// TwinCAT 3 PLC project PLC_Server_02
// ProgramVersion: 3.1.4023.0
// libraries:
//   Tc2_MC2, * (Beckhoff Automation GmbH)
//   Tc2_Standard, * (Beckhoff Automation GmbH)
//   Tc2_System, * (Beckhoff Automation GmbH)
//   Tc3_Module, * (Beckhoff Automation GmbH)
// project tree:
//   DUTs/ ST_Motor.TcDUT, ST_MotorCtrl.TcDUT
//   / GlobalTextList.TcGTLO, PlcTask.TcTTO, VISU_TASK.TcTTO
//   POUs/ FB_Math.TcPOU, MAIN.TcPOU
//   VISUs/ motor_status.TcVIS, VisualizationManager.TcVMO (not stored)
// real-time tasks:
//   TASK PlcTask: cycle T#10ms, priority 20, ADS port 350
//   TASK VISU_TASK: cycle T#200000us, priority 30, ADS port 351
// motion (NC):
//   TASK NC-Task 1 SAF: cycle T#2ms, priority 4, ADS port 501
//   TASK NC-Task 1 SVB: cycle T#10ms, priority 8, ADS port 511
//   AXIS Motor-0 (id 1)
//     OtherSettings: AllowMotionCmdToSlave=true
//     encoder EncType=1
//     drive DrvType=5
//       Analog: TorqueSetpointScale=10, ScaleFactorActTorque=0.1
//       TimeComp: TaskDelayCycles=1
//     controller CtrType=1
//       CtrPara: PriorControlFactor=1
//         Observer: BandWidth=20
//   AXIS Motor-1 (id 2)
//     OtherSettings: AllowMotionCmdToSlave=true
//     encoder EncType=1
//     drive DrvType=5
//       Analog: TorqueSetpointScale=10, ScaleFactorActTorque=0.1
//       TimeComp: TaskDelayCycles=1
//     controller CtrType=1
//       CtrPara: PriorControlFactor=1
//         Observer: BandWidth=20
//   AXIS Motor-2 (id 3)
//     OtherSettings: AllowMotionCmdToSlave=true
//     encoder EncType=1
//     drive DrvType=5
//       Analog: TorqueSetpointScale=10, ScaleFactorActTorque=0.1
//       TimeComp: TaskDelayCycles=1
//     controller CtrType=1
//       CtrPara: PriorControlFactor=1
//         Observer: BandWidth=20
//   AXIS Motor-3 (id 4)
//     OtherSettings: AllowMotionCmdToSlave=true
//     encoder EncType=1
//     drive DrvType=5
//       Analog: TorqueSetpointScale=10, ScaleFactorActTorque=0.1
//       TimeComp: TaskDelayCycles=1
//     controller CtrType=1
//       CtrPara: PriorControlFactor=1
//         Observer: BandWidth=20
//   AXIS Motor-4 (id 5)
//     OtherSettings: AllowMotionCmdToSlave=true
//     encoder EncType=1
//     drive DrvType=5
//       Analog: TorqueSetpointScale=10, ScaleFactorActTorque=0.1
//       TimeComp: TaskDelayCycles=1
//     controller CtrType=1
//       CtrPara: PriorControlFactor=1
//         Observer: BandWidth=20
// variable links:
//   PLC-Server-02/PLC-Server-02 Instance <-> NC-Task 1 SAF/Axes/Motor-0
//     PlcTask Inputs/MAIN.Motor[0].ref.NcToPlc <-> Outputs/ToPlc
//     PlcTask Outputs/MAIN.Motor[0].ref.PlcToNc <-> Inputs/FromPlc
//   PLC-Server-02/PLC-Server-02 Instance <-> NC-Task 1 SAF/Axes/Motor-1
//     PlcTask Inputs/MAIN.Motor[1].ref.NcToPlc <-> Outputs/ToPlc
//     PlcTask Outputs/MAIN.Motor[1].ref.PlcToNc <-> Inputs/FromPlc
//   PLC-Server-02/PLC-Server-02 Instance <-> NC-Task 1 SAF/Axes/Motor-2
//     PlcTask Inputs/MAIN.Motor[2].ref.NcToPlc <-> Outputs/ToPlc
//     PlcTask Outputs/MAIN.Motor[2].ref.PlcToNc <-> Inputs/FromPlc
//   PLC-Server-02/PLC-Server-02 Instance <-> NC-Task 1 SAF/Axes/Motor-3
//     PlcTask Inputs/MAIN.Motor[3].ref.NcToPlc <-> Outputs/ToPlc
//     PlcTask Outputs/MAIN.Motor[3].ref.PlcToNc <-> Inputs/FromPlc
//   PLC-Server-02/PLC-Server-02 Instance <-> NC-Task 1 SAF/Axes/Motor-4
//     PlcTask Inputs/MAIN.Motor[4].ref.NcToPlc <-> Outputs/ToPlc
//     PlcTask Outputs/MAIN.Motor[4].ref.PlcToNc <-> Inputs/FromPlc

CONFIGURATION PLC_Server_02
    RESOURCE PLC ON TwinCAT3
        TASK PlcTask(INTERVAL := T#10ms, PRIORITY := 20);
        TASK VISU_TASK(INTERVAL := T#200000us, PRIORITY := 30);
        PROGRAM MAIN WITH PlcTask : MAIN;
        PROGRAM VisuElems_Visu_Prg WITH VISU_TASK : VisuElems.Visu_Prg;
    END_RESOURCE
END_CONFIGURATION

// ---- DUTs/ST_Motor.TcDUT
TYPE ST_Motor :
STRUCT
	ref 	: AXIS_REF;
	fbPower : MC_Power;
	fbReset : MC_Reset;
	fbStop 	: MC_Stop;
	fbStart : MC_MoveVelocity;
	ctrl 	: ST_MotorCtrl;
	
END_STRUCT
END_TYPE

// ---- DUTs/ST_MotorCtrl.TcDUT
TYPE ST_MotorCtrl :
STRUCT
	power	: BOOL;
	start	: BOOL;
	stop	: BOOL;
	reset	: BOOL;
	velo 	: INT;
END_STRUCT
END_TYPE

// ---- POUs/MAIN.TcPOU
PROGRAM MAIN
VAR
{attribute 'OPC.UA.DA':='1'}	
	Motor : ARRAY [0..4] OF ST_Motor;
{attribute 'OPC.UA.DA':='1'}
	fbMath : ARRAY [0..4] OF FB_Math;
	
END_VAR

MAIN.aMotor_0();
MAIN.aMotor_1();
MAIN.aMotor_2();
MAIN.aMotor_3();
MAIN.aMotor_4();

ACTION aMotor_0:
// Motor 0 - Function Blocks ///////////////////////////////////////////////////////////

IF Motor[0].ctrl.velo > 2000 THEN
	Motor[0].ctrl.velo := 2000;
ELSIF Motor[0].ctrl.velo < 0 THEN
	Motor[0].ctrl.velo := 50;
END_IF

Motor[0].ref.ReadStatus();


Motor[0].fbPower(
	Axis:= Motor[0].ref, 
	Enable:= Motor[0].ctrl.power, 
	Enable_Positive:= Motor[0].ctrl.power, 
	Enable_Negative:= Motor[0].ctrl.power, 
	Status=> , 
	Busy=> , 
	Active=> , 
	Error=> , 
	ErrorID=>
	);
	
Motor[0].fbStart(
	Axis:= Motor[0].ref, 
	Execute:=  Motor[0].ctrl.start, 
	Velocity:=  Motor[0].ctrl.velo, 
	Acceleration:= 500, 
	Deceleration:= 500, 
	Jerk:= 1000, 
	InVelocity=> , 
	Busy=> , 
	Active=> , 
	CommandAborted=> , 
	Error=> , 
	ErrorID=> );
	
Motor[0].fbStop(
	Axis:= Motor[0].ref, 
	Execute:= Motor[0].ctrl.stop , 
	Deceleration:= 1000, 
	Jerk:= 1000, 
	Options:= , 
	Done=> , 
	Busy=> , 
	Active=> , 
	CommandAborted=> , 
	Error=> , 
	ErrorID=> );
	
Motor[0].fbReset(
	Axis:= Motor[0].ref, 
	Execute:= Motor[0].ctrl.reset, 
	Done=> , 
	Busy=> , 
	Error=> , 
	ErrorID=> );
END_ACTION

ACTION aMotor_1:
// Motor 1 - Function Blocks ///////////////////////////////////////////////////////////

IF Motor[1].ctrl.velo > 2000 THEN
	Motor[1].ctrl.velo := 2000;
ELSIF Motor[1].ctrl.velo < 0 THEN
	Motor[1].ctrl.velo := 50;
END_IF

Motor[1].ref.ReadStatus();


Motor[1].fbPower(
	Axis:= Motor[1].ref, 
	Enable:= Motor[1].ctrl.power, 
	Enable_Positive:= Motor[1].ctrl.power, 
	Enable_Negative:= Motor[1].ctrl.power, 
	Status=> , 
	Busy=> , 
	Active=> , 
	Error=> , 
	ErrorID=>
	);
	
Motor[1].fbStart(
	Axis:= Motor[1].ref, 
	Execute:=  Motor[1].ctrl.start, 
	Velocity:=  Motor[1].ctrl.velo, 
	Acceleration:= 500, 
	Deceleration:= 500, 
	Jerk:= 1000, 
	InVelocity=> , 
	Busy=> , 
	Active=> , 
	CommandAborted=> , 
	Error=> , 
	ErrorID=> );
	
Motor[1].fbStop(
	Axis:= Motor[1].ref, 
	Execute:= Motor[1].ctrl.stop , 
	Deceleration:= 1000, 
	Jerk:= 1000, 
	Options:= , 
	Done=> , 
	Busy=> , 
	Active=> , 
	CommandAborted=> , 
	Error=> , 
	ErrorID=> );
	
Motor[1].fbReset(
	Axis:= Motor[1].ref, 
	Execute:= Motor[1].ctrl.reset, 
	Done=> , 
	Busy=> , 
	Error=> , 
	ErrorID=> );
END_ACTION

ACTION aMotor_2:
// Motor 2 - Function Blocks ///////////////////////////////////////////////////////////

IF Motor[2].ctrl.velo > 2000 THEN
	Motor[2].ctrl.velo := 2000;
ELSIF Motor[2].ctrl.velo < 0 THEN
	Motor[2].ctrl.velo := 50;
END_IF

Motor[2].ref.ReadStatus();


Motor[2].fbPower(
	Axis:= Motor[2].ref, 
	Enable:= Motor[2].ctrl.power, 
	Enable_Positive:= Motor[2].ctrl.power, 
	Enable_Negative:= Motor[2].ctrl.power, 
	Status=> , 
	Busy=> , 
	Active=> , 
	Error=> , 
	ErrorID=>
	);
	
Motor[2].fbStart(
	Axis:= Motor[2].ref, 
	Execute:=  Motor[2].ctrl.start, 
	Velocity:=  Motor[2].ctrl.velo, 
	Acceleration:= 500, 
	Deceleration:= 500, 
	Jerk:= 1000, 
	InVelocity=> , 
	Busy=> , 
	Active=> , 
	CommandAborted=> , 
	Error=> , 
	ErrorID=> );
	
Motor[2].fbStop(
	Axis:= Motor[2].ref, 
	Execute:= Motor[2].ctrl.stop , 
	Deceleration:= 1000, 
	Jerk:= 1000, 
	Options:= , 
	Done=> , 
	Busy=> , 
	Active=> , 
	CommandAborted=> , 
	Error=> , 
	ErrorID=> );
	
Motor[2].fbReset(
	Axis:= Motor[2].ref, 
	Execute:= Motor[2].ctrl.reset, 
	Done=> , 
	Busy=> , 
	Error=> , 
	ErrorID=> );
END_ACTION

ACTION aMotor_3:
// Motor 3 - Function Blocks ///////////////////////////////////////////////////////////

IF Motor[3].ctrl.velo > 2000 THEN
	Motor[3].ctrl.velo := 2000;
ELSIF Motor[3].ctrl.velo < 0 THEN
	Motor[3].ctrl.velo := 50;
END_IF

Motor[3].ref.ReadStatus();


Motor[3].fbPower(
	Axis:= Motor[3].ref, 
	Enable:= Motor[3].ctrl.power, 
	Enable_Positive:= Motor[3].ctrl.power, 
	Enable_Negative:= Motor[3].ctrl.power, 
	Status=> , 
	Busy=> , 
	Active=> , 
	Error=> , 
	ErrorID=>
	);
	
Motor[3].fbStart(
	Axis:= Motor[3].ref, 
	Execute:=  Motor[3].ctrl.start, 
	Velocity:=  Motor[3].ctrl.velo, 
	Acceleration:= 500, 
	Deceleration:= 500, 
	Jerk:= 1000, 
	InVelocity=> , 
	Busy=> , 
	Active=> , 
	CommandAborted=> , 
	Error=> , 
	ErrorID=> );
	
Motor[3].fbStop(
	Axis:= Motor[3].ref, 
	Execute:= Motor[3].ctrl.stop , 
	Deceleration:= 1000, 
	Jerk:= 1000, 
	Options:= , 
	Done=> , 
	Busy=> , 
	Active=> , 
	CommandAborted=> , 
	Error=> , 
	ErrorID=> );
	
Motor[3].fbReset(
	Axis:= Motor[3].ref, 
	Execute:= Motor[3].ctrl.reset, 
	Done=> , 
	Busy=> , 
	Error=> , 
	ErrorID=> );
END_ACTION

ACTION aMotor_4:
// Motor 4 - Function Blocks ///////////////////////////////////////////////////////////

IF Motor[4].ctrl.velo > 2000 THEN
	Motor[4].ctrl.velo := 2000;
ELSIF Motor[4].ctrl.velo < 0 THEN
	Motor[4].ctrl.velo := 50;
END_IF

Motor[4].ref.ReadStatus();


Motor[4].fbPower(
	Axis:= Motor[4].ref, 
	Enable:= Motor[4].ctrl.power, 
	Enable_Positive:= Motor[4].ctrl.power, 
	Enable_Negative:= Motor[4].ctrl.power, 
	Status=> , 
	Busy=> , 
	Active=> , 
	Error=> , 
	ErrorID=>
	);
	
Motor[4].fbStart(
	Axis:= Motor[4].ref, 
	Execute:=  Motor[4].ctrl.start, 
	Velocity:=  Motor[4].ctrl.velo, 
	Acceleration:= 500, 
	Deceleration:= 500, 
	Jerk:= 1000, 
	InVelocity=> , 
	Busy=> , 
	Active=> , 
	CommandAborted=> , 
	Error=> , 
	ErrorID=> );
	
Motor[4].fbStop(
	Axis:= Motor[4].ref, 
	Execute:= Motor[4].ctrl.stop , 
	Deceleration:= 1000, 
	Jerk:= 1000, 
	Options:= , 
	Done=> , 
	Busy=> , 
	Active=> , 
	CommandAborted=> , 
	Error=> , 
	ErrorID=> );
	
Motor[4].fbReset(
	Axis:= Motor[4].ref, 
	Execute:= Motor[4].ctrl.reset, 
	Done=> , 
	Busy=> , 
	Error=> , 
	ErrorID=> );
END_ACTION

END_PROGRAM

// ---- POUs/FB_Math.TcPOU
FUNCTION_BLOCK FB_Math
VAR_INPUT
END_VAR
VAR_OUTPUT
END_VAR
VAR
	{attribute 'OPC.UA.DA':='1'}
	nNumberOfCallsMMul : INT;
	{attribute 'OPC.UA.DA':='1'}
	nNumberOfCallsMAdd : INT;
	{attribute 'OPC.UA.DA':='1'}
	nNumberOfCallsMRpm : INT;
END_VAR

{attribute 'TcRpcEnable':='1'}
METHOD M_Add : DINT
VAR_INPUT
	a : INT;
	b : INT;
END_VAR
M_Add := a + b;
nNumberOfCallsMAdd := nNumberOfCallsMAdd + 1;
END_METHOD

{attribute 'TcRpcEnable':='1'}
METHOD M_Mul : DINT
VAR_INPUT
	a : INT;
	b : INT;
END_VAR
M_Mul := a * b;
nNumberOfCallsMMul := nNumberOfCallsMMul + 1;
END_METHOD

{attribute 'TcRpcEnable':='1'}
METHOD M_Rpm : DINT
VAR_INPUT
	motorSpeed : DINT;
	gearboxRatio : DINT;
END_VAR
M_Rpm := motorSpeed/gearboxRatio;
nNumberOfCallsMRpm := nNumberOfCallsMRpm + 1;
END_METHOD

END_FUNCTION_BLOCK

// ---- GlobalTextList.TcGTLO
TEXTLIST GlobalTextList
  525 = 'Motor 0 - Enabled'
  403 = 'Motor 0 - Error'
  824 = 'Motor 0 - Running'
  748 = 'Motor 0 - Speed'
  648 = 'Motor 0 - Stopping'
  957 = 'Motor 1 - Enabled'
  496 = 'Motor 1 - Error'
  215 = 'Motor 1 - Running'
  878 = 'Motor 1 - Speed'
  666 = 'Motor 1 - Stopping'
  520 = 'Motor 2 - Enabled'
  864 = 'Motor 2 - Error'
  650 = 'Motor 2 - Running'
  966 = 'Motor 2 - Speed'
  229 = 'Motor 2 - Stopping'
  281 = 'Motor 3 - Enabled'
  99 = 'Motor 3 - Error'
  861 = 'Motor 3 - Running'
  669 = 'Motor 3 - Speed'
  621 = 'Motor 3 - Stopping'
  685 = 'Motor 4 - Enabled'
  400 = 'Motor 4 - Error'
  1 = 'Motor 4 - Running'
  509 = 'Motor 4 - Speed'
  862 = 'Motor 4 - Stopping'
  780 = 'Motor 5 - Running'
END_TEXTLIST

// ---- VISUs/motor_status.TcVIS
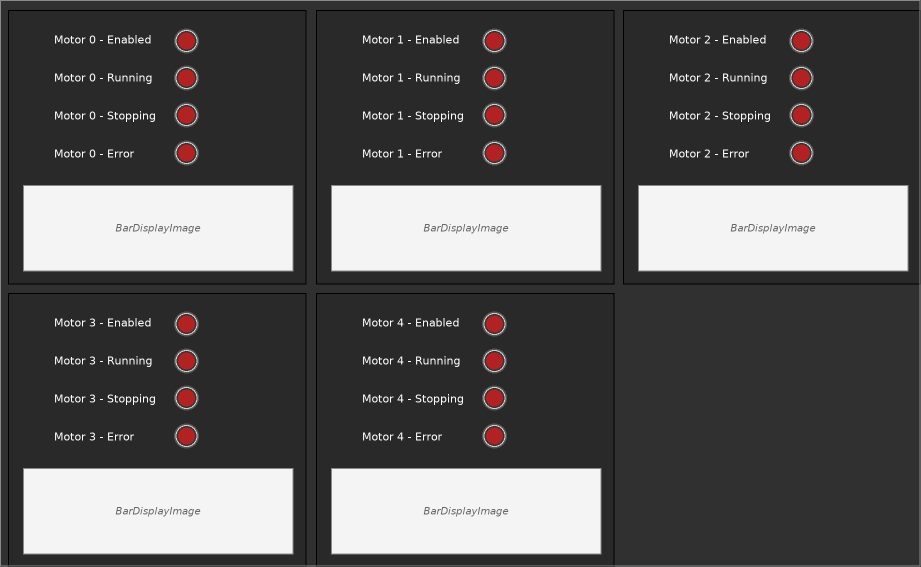
VISUALIZATION motor_status  // 921x567
    Rectangle (8,10 298x274)
    Label (51,25 150x30), "Motor 0 - Enabled"
    BarDisplayImage (23,185 270x86), value: MAIN.Motor[0].ref.NcToPlc.ActVelo, style: BarDisplayImage-Gray, scale format: %.1f, scale 0..2000
        p518627256: Motor 0 - Speed
    Lamp1 (172,26 29x30), variable: MAIN.Motor[0].fbPower.Status, style: Lamp-Lamp1-Red
    Label (51,63 150x30), "Motor 0 - Running"
    Label (51,101 150x30), "Motor 0 - Stopping"
    Label (51,139 150x30), "Motor 0 - Error"
    Lamp1 (172,63 29x30), variable: MAIN.Motor[0].ref.Status.Moving, style: Lamp-Lamp1-Red
    Lamp1 (172,100 29x30), variable: MAIN.Motor[0].ref.Status.Stopping, style: Lamp-Lamp1-Red
    Lamp1 (172,138 29x30), variable: MAIN.Motor[0].ref.Status.Error, style: Lamp-Lamp1-Red
    Rectangle (316,10 298x274)
    Label (359,25 150x30), "Motor 1 - Enabled"
    BarDisplayImage (331,185 270x86), value: MAIN.Motor[1].ref.NcToPlc.ActVelo, style: BarDisplayImage-Gray, scale format: %.1f, scale 0..2000
        p518627256: Motor 1 - Speed
    Lamp1 (480,26 29x30), variable: MAIN.Motor[1].fbPower.Status, style: Lamp-Lamp1-Red
    Label (359,63 150x30), "Motor 1 - Running"
    Label (359,101 150x30), "Motor 1 - Stopping"
    Label (359,139 150x30), "Motor 1 - Error"
    Lamp1 (480,63 29x30), variable: MAIN.Motor[1].ref.Status.Moving, style: Lamp-Lamp1-Red
    Lamp1 (480,100 29x30), variable: MAIN.Motor[1].ref.Status.Stopping, style: Lamp-Lamp1-Red
    Lamp1 (480,138 29x30), variable: MAIN.Motor[1].ref.Status.Error, style: Lamp-Lamp1-Red
    Rectangle (623,10 298x274)
    Label (666,25 150x30), "Motor 2 - Enabled"
    BarDisplayImage (638,185 270x86), value: MAIN.Motor[2].ref.NcToPlc.ActVelo, style: BarDisplayImage-Gray, scale format: %.1f, scale 0..2000
        p518627256: Motor 2 - Speed
    Lamp1 (787,26 29x30), variable: MAIN.Motor[2].fbPower.Status, style: Lamp-Lamp1-Red
    Label (666,63 150x30), "Motor 2 - Running"
    Label (666,101 150x30), "Motor 2 - Stopping"
    Label (666,139 150x30), "Motor 2 - Error"
    Lamp1 (787,63 29x30), variable: MAIN.Motor[2].ref.Status.Moving, style: Lamp-Lamp1-Red
    Lamp1 (787,100 29x30), variable: MAIN.Motor[2].ref.Status.Stopping, style: Lamp-Lamp1-Red
    Lamp1 (787,138 29x30), variable: MAIN.Motor[2].ref.Status.Error, style: Lamp-Lamp1-Red
    Rectangle (8,293 298x274)
    Label (51,308 150x30), "Motor 3 - Enabled"
    BarDisplayImage (23,468 270x86), value: MAIN.Motor[3].ref.NcToPlc.ActVelo, style: BarDisplayImage-Gray, scale format: %.1f, scale 0..2000
        p518627256: Motor 3 - Speed
    Lamp1 (172,309 29x30), variable: MAIN.Motor[3].fbPower.Status, style: Lamp-Lamp1-Red
    Label (51,346 150x30), "Motor 3 - Running"
    Label (51,384 150x30), "Motor 3 - Stopping"
    Label (51,422 150x30), "Motor 3 - Error"
    Lamp1 (172,346 29x30), variable: MAIN.Motor[3].ref.Status.Moving, style: Lamp-Lamp1-Red
    Lamp1 (172,383 29x30), variable: MAIN.Motor[3].ref.Status.Stopping, style: Lamp-Lamp1-Red
    Lamp1 (172,421 29x30), variable: MAIN.Motor[3].ref.Status.Error, style: Lamp-Lamp1-Red
    Rectangle (316,293 298x274)
    Label (359,308 150x30), "Motor 4 - Enabled"
    BarDisplayImage (331,468 270x86), value: MAIN.Motor[4].ref.NcToPlc.ActVelo, style: BarDisplayImage-Gray, scale format: %.1f, scale 0..2000
        p518627256: Motor 4 - Speed
    Lamp1 (480,309 29x30), variable: MAIN.Motor[4].fbPower.Status, style: Lamp-Lamp1-Red
    Label (359,346 150x30), "Motor 4 - Running"
    Label (359,384 150x30), "Motor 4 - Stopping"
    Label (359,422 150x30), "Motor 4 - Error"
    Lamp1 (480,346 29x30), variable: MAIN.Motor[4].ref.Status.Moving, style: Lamp-Lamp1-Red
    Lamp1 (480,383 29x30), variable: MAIN.Motor[4].ref.Status.Stopping, style: Lamp-Lamp1-Red
    Lamp1 (480,421 29x30), variable: MAIN.Motor[4].ref.Status.Error, style: Lamp-Lamp1-Red
END_VISUALIZATION
